// TIA Portal project "1513_Buch_Plenk_2_WWW" (V13)

(* hardware
DEVICE "S71500/ET200MP-Station_1"  S7-1500 station
   slot 0: "Profilschiene_0"  6ES7 590-1***0-0AA0
   slot 1: "PLC_1"  CPU 1513-1 PN  6ES7 513-1AL00-0AB0  V1.8
DEVICE "HMI_1"  TP1500 Basic color PN
   slot 0: "HMI"  HMI  6AV6 647-0AG11-3AX0  12.0.0.0
   slot 1: "HMI_RT_1"  TP1500 Basic color PN  6AV6 647-0AG11-3AX0  12.0.0.0
   slot 5: "HMI_1.IE_CP_1"  PROFINET Schnittstelle
      slot 1: "PROFINET Schnittstelle_1"  PROFINET Schnittstelle
         slot 1: "Port_1"  Port
*)

// ===== PLC "PLC_1"  CPU 1513-1 PN =====

VAR_GLOBAL   // PLC tag table "Standard-Variablentabelle"
   "System_Byte" AT %MB1 : Byte;
   "FirstScan" AT %M1.0 : Bool;
   "DiagStatusUpdate" AT %M1.1 : Bool;
   "AlwaysTRUE" AT %M1.2 : Bool;
   "AlwaysFALSE" AT %M1.3 : Bool;
   "Clock_Byte" AT %MB0 : Byte;
   "Clock_10Hz" AT %M0.0 : Bool;
   "Clock_5Hz" AT %M0.1 : Bool;
   "Clock_2.5Hz" AT %M0.2 : Bool;
   "Clock_2Hz" AT %M0.3 : Bool;
   "Clock_1.25Hz" AT %M0.4 : Bool;
   "Clock_1Hz" AT %M0.5 : Bool;
   "Clock_0.625Hz" AT %M0.6 : Bool;
   "Clock_0.5Hz" AT %M0.7 : Bool;
   "Setzen" AT %M2.0 : Bool;
   "Ruecksetzen" AT %M2.1 : Bool;
   "Vorbelegung" AT %MW4 : Int;
   "Zaehlwert" AT %MW6 : Int;
   "Eingabewert" AT %MW8 : Int;
   "Fehlercode" AT %MW10 : Int;
END_VAR

// folder: System blocks/Program resources

DATA_BLOCK "IEC_Counter_0_DB"   // DB1
{ S7_Optimized_Access := 'FALSE' }
AUTHOR : Simatic
FAMILY : IEC
NAME : CNTR
VERSION : 1.0
// stored: InstanceOfName ?
"?"
BEGIN
END_DATA_BLOCK

// folder: (top level)

ORGANIZATION_BLOCK "Main"   // OB1, FBD, ProgramCycle
TITLE = "Main Program Sweep (Cycle)"
{ S7_Optimized_Access := 'FALSE' }
VERSION : 0.1
BEGIN

REGION Network 1
   // Der Startwert für den Zähler wird gesetzt (in den Zähler-DB schreiben)
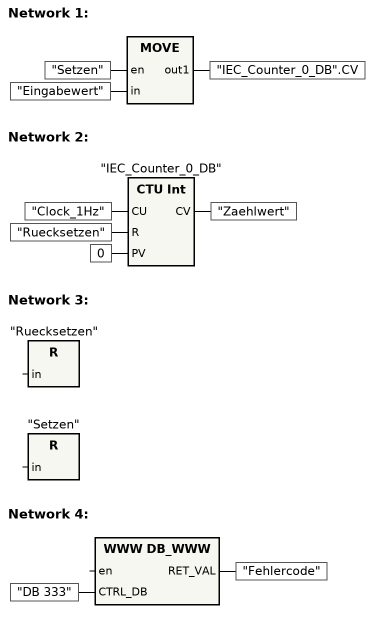
   IF "Setzen" THEN "IEC_Counter_0_DB".CV := "Eingabewert"; END_IF;
END_REGION

REGION Network 2
   // Der IEC-Vorwärtszähler wird im 1-Sekunden Takt hochgezählt; die Zählwertausgabe erfolgt in eine INT-Variable
   "IEC_Counter_0_DB".CTU(CU := "Clock_1Hz", R := "Ruecksetzen", PV := 0, CV => "Zaehlwert");
END_REGION

REGION Network 3
   // Die von der Webseite aus gesteuerten Merker wieder rücksetzen
   "Ruecksetzen" := FALSE;
   "Setzen" := FALSE;
END_REGION

REGION Network 4
   // Anwender-Webseiten mit dem Programm in der CPU synchronisieren - WWW muss  im zyklischen Programmteil stehen
   "Fehlercode" := WWW(CTRL_DB := "DB 333");
END_REGION
END_ORGANIZATION_BLOCK